TYPE A_Devices : INT(1..3); END_TYPE

(* stored: Version 1.1.0.1
   DUT A_Devices: Id {31ebb4fe-c07f-4e6e-aebe-f3907e471ed3} *)
